# EPICS StreamDevice protocol: SSABoosterSup/SSABooster.proto
getData {
    ReplyTimeout=1000;
    ReadTimeout=100;
    separator=';';
    InTerminator=CR, LF;
    ExtraInput=Ignore;
    out "\$1";
    in  "%8s";
}
